PROGRAM MAIN
VAR
	fbSH200A : FB_Simplex();
END_VAR

fbSH200A.M_Jog();
//fbSH200A.M_LogValues();
SerialCommunication();
//fbSH200A();

END_PROGRAM

(* stored: Version 1.1.0.1, ProductVersion 3.1.4020.12
   POU MAIN: Id {a6f35caf-0754-4117-99e9-4db78ebe9f31}, SpecialFunc None *)
